Staubli VAL3: writeIntValue.pgx

public program writeIntValue(num handle_, num col_, num row_, num value_, bool& result_[])
  local string strCell
begin
  // write an integer value into a cell
  nCommand[handle_]=coSI
  call coord2Cell(col_,row_,strCell)
  call sendCommand(handle_,"si"+strCell+toString("0.0",roundDown(value_)),result_)
end
